FUNCTION_BLOCK E_SPLIT_3 (* Composite Function Block Type *)
  (* Standard: 61499-2 *)
  (* Version 0.0, 9/22/2026, macie, Schneider Electric, template *)
  PACKAGE Main;
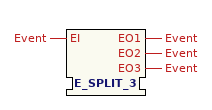
  EVENT_INPUT
    EI; (* Initialization Request *)
  END_EVENT
  EVENT_OUTPUT
    EO1; (* Initialization Confirm *)
    EO2; (* Execution Confirmation *)
    EO3;
  END_EVENT
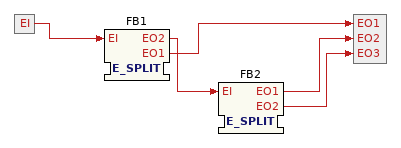
  FBS
    FB1 : E_SPLIT;
    FB2 : E_SPLIT;
  END_FBS
  EVENT_CONNECTIONS
    EI TO FB1.EI;
    FB1.EO2 TO FB2.EI;
    FB1.EO1 TO EO1;
    FB2.EO1 TO EO2;
    FB2.EO2 TO EO3;
  END_CONNECTIONS
END_FUNCTION_BLOCK
